              Waypoint Sacar_P2: TCP in base x=-1173.973 y=-367.221 z=3.618 mm, rx=2.0094 ry=-2.4021 rz=-0.0129 rad; joints [10.662, -31.588, 47.899, -16.562, 101.711, 0.111] deg
            Wait Sleep waitTime=0.5
            MoveDirectionNode (selectedDirection=YPlus toolParams=0.0013, 2.0E-4)
              Until TOOL_CONTACT_DETECTION (allowActions=false retraction=0 decelerationAcceleration=9 decelerationAngularAcceleration=34.906585)
            Wait Sleep waitTime=2
            P2 := pose_add(get_actual_tcp_pose(), P2)
            muestrasTomadas := muestrasTomadas+1
          muestrasTomadas := 0
          var_1 := (P2[0])/muestras
          var_2 := (P2[1])/muestras
          rotaciones := get_actual_tcp_pose()
          var_3 := rotaciones[3]
          var_4 := rotaciones[4]
          var_5 := rotaciones[5]
          P2 := p[var_1,var_2,-0.37,var_3,var_4,var_5]
        MoveJ speed 60 deg/s, acceleration 80 deg/s^2 (useActiveTCP=true) feature=Base
          Waypoint Casa2: TCP in base x=-771.144 y=-432.919 z=130.536 mm, rx=2.0101 ry=-2.4029 rz=-0.0102 rad; joints [21.813, -67.428, 96.538, -29.271, 112.826, 0.127] deg
        Folder m1
          var_1 := (P1[0])
          var_2 := (P1[1])
          var_3 := (P2[0])
          var_4 := (P2[1])
          m1 := (var_4-var_2)/(var_3-var_1)
        Folder b1
          b1 := ((m1*var_1)-var_2)*(-1)
        MoveJ speed 60 deg/s, acceleration 80 deg/s^2 (useActiveTCP=true) feature=Base
          Waypoint Casa1: TCP in base x=-416.709 y=-228.23 z=81.827 mm, rx=2.012 ry=-2.4053 rz=-0.0107 rad; joints [11.287, -103.558, 142.129, -38.591, 102.295, 0.04] deg
        Folder P3
          Loop While (checkContinuously=false) expression=muestrasTomadas<muestras
            MoveJ speed 60 deg/s, acceleration 80 deg/s^2 (useActiveTCP=true) feature=Base
              Waypoint Sacar_P3: motionParameters(jointSpeed=1.047198 jointAcceleration=1.396263 cartesianSpeed=0.1 cartesianAcceleration=0.15); TCP in base x=-387.702 y=-99.027 z=-5.945 mm, rx=2.01 ry=-2.4029 rz=-0.0102 rad; joints [-19.937, -108.067, 157.062, -49.107, 71.061, 0.231] deg
            Wait Sleep waitTime=0.5
            MoveDirectionNode (selectedDirection=XPlus toolParams=0.0013, 2.0E-4)
              Until TOOL_CONTACT_DETECTION (allowActions=false retraction=0 decelerationAcceleration=9 decelerationAngularAcceleration=34.906585)
            Wait Sleep waitTime=2
            P3 := pose_add(get_actual_tcp_pose(), P3)
            muestrasTomadas := muestrasTomadas+1
          muestrasTomadas := 0
          var_1 := (P3[0])/muestras
          var_2 := (P3[1])/muestras
          rotaciones := get_actual_tcp_pose()
          var_3 := rotaciones[3]
          var_4 := rotaciones[4]
          var_5 := rotaciones[5]
          P3 := p[var_1,var_2,-0.37,var_3,var_4,var_5]
        MoveJ speed 60 deg/s, acceleration 80 deg/s^2 (useActiveTCP=true) feature=Base
          Waypoint Casa1: TCP in base x=-416.709 y=-228.23 z=81.827 mm, rx=2.012 ry=-2.4053 rz=-0.0107 rad; joints [11.287, -103.558, 142.129, -38.591, 102.295, 0.04] deg
        Folder P4
          Loop While (checkContinuously=false) expression=muestrasTomadas<muestras
            MoveJ speed 60 deg/s, acceleration 80 deg/s^2 (useActiveTCP=true) feature=Base
              Waypoint Sacar_P4: motionParameters(jointSpeed=1.047198 jointAcceleration=1.396263 cartesianSpeed=0.1 cartesianAcceleration=0.15); TCP in base x=-386.694 y=-336.624 z=-4.009 mm, rx=2.0101 ry=-2.4029 rz=-0.0102 rad; joints [30.346, -87.141, 140.524, -53.547, 121.328, 0.136] deg
            Wait Sleep waitTime=0.5
            MoveDirectionNode (selectedDirection=XPlus toolParams=0.0013, 2.0E-4)
              Until TOOL_CONTACT_DETECTION (allowActions=false retraction=0 decelerationAcceleration=9 decelerationAngularAcceleration=34.906585)
            Wait Sleep waitTime=2
            P4 := pose_add(get_actual_tcp_pose(), P4)
            muestrasTomadas := muestrasTomadas+1
          muestrasTomadas := 0
          var_1 := (P4[0])/muestras
          var_2 := (P4[1])/muestras
          rotaciones := get_actual_tcp_pose()
          var_3 := rotaciones[3]
          var_4 := rotaciones[4]
          var_5 := rotaciones[5]
          P4 := p[var_1,var_2,-0.37,var_3,var_4,var_5]
        MoveJ speed 60 deg/s, acceleration 80 deg/s^2 (useActiveTCP=true) feature=Base
          Waypoint Casa1: TCP in base x=-416.709 y=-228.23 z=81.827 mm, rx=2.012 ry=-2.4053 rz=-0.0107 rad; joints [11.287, -103.558, 142.129, -38.591, 102.295, 0.04] deg
        Folder m2
          var_1 := (P3[0])
          var_2 := (P3[1])
          var_3 := (P4[0])
          var_4 := (P4[1])
          m2 := (var_4-var_2)/(var_3-var_1)
        Folder b2
          b2 := ((m2*var_1)-var_2)*(-1)
        Folder Xd y Yd
          Xd := (b2-b1)/(m1-m2)
          Yd := (m1*Xd)+b1
        Folder Xp y Yp
          Xp := (1)/(sqrt((m1*m1)+1))
          Yp := (m2)/(sqrt((m2*m2)+1))
        Folder Origen
          Xfin := ((0*Xp)-(Xd)-(0*(1/m2)))*(-1)
          Yfin := ((0*Yp)-(Yd)+(0*m1))*(-1)
          rotaciones := get_actual_tcp_pose()
          var_3 := rotaciones[3]
          var_4 := rotaciones[4]
          var_5 := rotaciones[5]
          PosFinal := p[Xfin+0.00208915,Yfin+0.00208915,0.11,var_3,var_4,var_5]
          origen := PosFinal
        MoveJ speed 60 deg/s, acceleration 80 deg/s^2 (useActiveTCP=true) feature=Base
          Waypoint Waypoint (Variable): motionParameters(jointSpeed=1.047198 jointAcceleration=1.396263 cartesianSpeed=0.15 cartesianAcceleration=0.2); variable=PosFinal
        MoveDirectionNode (selectedDirection=ZPlus)
          Until DISTANCE (allowActions=false deceleration=3 distanceNodeType=STOP) Distance=0.1; motionParameters(blendRadius=0)
        MoveJ speed 60 deg/s, acceleration 80 deg/s^2 (useActiveTCP=true) feature=Base
          Waypoint Casa2: TCP in base x=-771.144 y=-432.919 z=130.536 mm, rx=2.0101 ry=-2.4029 rz=-0.0102 rad; joints [21.813, -67.428, 96.538, -29.271, 112.826, 0.127] deg
        Folder Linea1
          SuppressedNode
            Folder Buje1
              Xfin := ((0.09525*Xp)-(Xd)-(-0.0127*(1/m2)))*(-1)
              Yfin := ((-0.0127*Yp)-(Yd)+(0.09525*m1))*(-1)
              rotaciones := get_actual_tcp_pose()
              var_3 := rotaciones[3]
              var_4 := rotaciones[4]
              var_5 := rotaciones[5]
              PosFinal := p[Xfin+0.00208915,Yfin+0.00208915,0.03,var_3,var_4,var_5]
              MoveL speed 250 mm/s, acceleration 1200 mm/s^2 (useActiveTCP=true) feature=Base
                MoveJ speed 60 deg/s, acceleration 80 deg/s^2 (useActiveTCP=true) feature=Base
                  Waypoint Waypoint (Variable): motionParameters(jointSpeed=1.047198 jointAcceleration=1.396263 cartesianSpeed=0.15 cartesianAcceleration=0.2); variable=PosFinal
                MoveDirectionNode (selectedDirection=ZMinus toolParams=0.02, 0.02)
                  Until DISTANCE (allowActions=false deceleration=3 distanceNodeType=STOP) Distance=0.035; motionParameters(blendRadius=0)
                MoveDirectionNode (selectedDirection=ZPlus toolParams=0.02, 0.02)
                  Until DISTANCE (allowActions=false deceleration=3 distanceNodeType=STOP) Distance=0.035; motionParameters(blendRadius=0)
          SuppressedNode
            Folder Buje2
              Xfin := ((0.12065*Xp)-(Xd)-(-0.0127*(1/m2)))*(-1)
              Yfin := ((-0.0127*Yp)-(Yd)+(0.12065*m1))*(-1)
              rotaciones := get_actual_tcp_pose()
              var_3 := rotaciones[3]
              var_4 := rotaciones[4]
              var_5 := rotaciones[5]
              PosFinal := p[Xfin+0.00208915,Yfin+0.00208915,0.03,var_3,var_4,var_5]
              MoveL speed 250 mm/s, acceleration 1200 mm/s^2 (useActiveTCP=true) feature=Base
                MoveJ speed 60 deg/s, acceleration 80 deg/s^2 (useActiveTCP=true) feature=Base
                  Waypoint Waypoint (Variable): motionParameters(jointSpeed=1.047198 jointAcceleration=1.396263 cartesianSpeed=0.15 cartesianAcceleration=0.2); variable=PosFinal
                MoveDirectionNode (selectedDirection=ZMinus toolParams=0.02, 0.02)
                  Until DISTANCE (allowActions=false deceleration=3 distanceNodeType=STOP) Distance=0.035; motionParameters(blendRadius=0)
                MoveDirectionNode (selectedDirection=ZPlus toolParams=0.02, 0.02)
                  Until DISTANCE (allowActions=false deceleration=3 distanceNodeType=STOP) Distance=0.035; motionParameters(blendRadius=0)
          SuppressedNode
            Folder Buje3
              Xfin := ((0.14605*Xp)-(Xd)-(-0.0127*(1/m2)))*(-1)
              Yfin := ((-0.0127*Yp)-(Yd)+(0.14605*m1))*(-1)
              rotaciones := get_actual_tcp_pose()
              var_3 := rotaciones[3]
              var_4 := rotaciones[4]
              var_5 := rotaciones[5]
              PosFinal := p[Xfin+0.00208915,Yfin+0.00208915,0.03,var_3,var_4,var_5]
              MoveL speed 250 mm/s, acceleration 1200 mm/s^2 (useActiveTCP=true) feature=Base
                MoveJ speed 60 deg/s, acceleration 80 deg/s^2 (useActiveTCP=true) feature=Base
                  Waypoint Waypoint (Variable): motionParameters(jointSpeed=1.047198 jointAcceleration=1.396263 cartesianSpeed=0.15 cartesianAcceleration=0.2); variable=PosFinal
                MoveDirectionNode (selectedDirection=ZMinus toolParams=0.02, 0.02)
                  Until DISTANCE (allowActions=false deceleration=3 distanceNodeType=STOP) Distance=0.035; motionParameters(blendRadius=0)
                MoveDirectionNode (selectedDirection=ZPlus toolParams=0.02, 0.02)
                  Until DISTANCE (allowActions=false deceleration=3 distanceNodeType=STOP) Distance=0.035; motionParameters(blendRadius=0)
          SuppressedNode
            Folder Buje4
              Xfin := ((0.17145*Xp)-(Xd)-(-0.0127*(1/m2)))*(-1)
              Yfin := ((-0.0127*Yp)-(Yd)+(0.17145*m1))*(-1)
              rotaciones := get_actual_tcp_pose()
              var_3 := rotaciones[3]
              var_4 := rotaciones[4]
              var_5 := rotaciones[5]
              PosFinal := p[Xfin+0.00208915,Yfin+0.00208915,0.03,var_3,var_4,var_5]
              MoveL speed 250 mm/s, acceleration 1200 mm/s^2 (useActiveTCP=true) feature=Base
                MoveJ speed 60 deg/s, acceleration 80 deg/s^2 (useActiveTCP=true) feature=Base
                  Waypoint Waypoint (Variable): motionParameters(jointSpeed=1.047198 jointAcceleration=1.396263 cartesianSpeed=0.15 cartesianAcceleration=0.2); variable=PosFinal
                MoveDirectionNode (selectedDirection=ZMinus toolParams=0.02, 0.02)
                  Until DISTANCE (allowActions=false deceleration=3 distanceNodeType=STOP) Distance=0.035; motionParameters(blendRadius=0)
                MoveDirectionNode (selectedDirection=ZPlus toolParams=0.02, 0.02)
                  Until DISTANCE (allowActions=false deceleration=3 distanceNodeType=STOP) Distance=0.035; motionParameters(blendRadius=0)
          SuppressedNode
            Folder Buje5
              Xfin := ((0.19685*Xp)-(Xd)-(-0.0127*(1/m2)))*(-1)
              Yfin := ((-0.0127*Yp)-(Yd)+(0.19685*m1))*(-1)
              rotaciones := get_actual_tcp_pose()
              var_3 := rotaciones[3]
              var_4 := rotaciones[4]
              var_5 := rotaciones[5]
              PosFinal := p[Xfin+0.00208915,Yfin+0.00208915,0.03,var_3,var_4,var_5]
              MoveL speed 250 mm/s, acceleration 1200 mm/s^2 (useActiveTCP=true) feature=Base
                MoveJ speed 60 deg/s, acceleration 80 deg/s^2 (useActiveTCP=true) feature=Base
                  Waypoint Waypoint (Variable): motionParameters(jointSpeed=1.047198 jointAcceleration=1.396263 cartesianSpeed=0.15 cartesianAcceleration=0.2); variable=PosFinal
                MoveDirectionNode (selectedDirection=ZMinus toolParams=0.02, 0.02)
                  Until DISTANCE (allowActions=false deceleration=3 distanceNodeType=STOP) Distance=0.035; motionParameters(blendRadius=0)
                MoveDirectionNode (selectedDirection=ZPlus toolParams=0.02, 0.02)
                  Until DISTANCE (allowActions=false deceleration=3 distanceNodeType=STOP) Distance=0.035; motionParameters(blendRadius=0)
          SuppressedNode
            Folder Buje6
              Xfin := ((0.22225*Xp)-(Xd)-(-0.0127*(1/m2)))*(-1)
              Yfin := ((-0.0127*Yp)-(Yd)+(0.22225*m1))*(-1)
              rotaciones := get_actual_tcp_pose()
              var_3 := rotaciones[3]
              var_4 := rotaciones[4]
              var_5 := rotaciones[5]
              PosFinal := p[Xfin+0.00208915,Yfin+0.00208915,0.03,var_3,var_4,var_5]
              MoveL speed 250 mm/s, acceleration 1200 mm/s^2 (useActiveTCP=true) feature=Base
                MoveJ speed 60 deg/s, acceleration 80 deg/s^2 (useActiveTCP=true) feature=Base
                  Waypoint Waypoint (Variable): motionParameters(jointSpeed=1.047198 jointAcceleration=1.396263 cartesianSpeed=0.15 cartesianAcceleration=0.2); variable=PosFinal
                MoveDirectionNode (selectedDirection=ZMinus toolParams=0.02, 0.02)
                  Until DISTANCE (allowActions=false deceleration=3 distanceNodeType=STOP) Distance=0.035; motionParameters(blendRadius=0)
                MoveDirectionNode (selectedDirection=ZPlus toolParams=0.02, 0.02)
                  Until DISTANCE (allowActions=false deceleration=3 distanceNodeType=STOP) Distance=0.035; motionParameters(blendRadius=0)
          SuppressedNode
            Folder Buje7
              Xfin := ((0.24765*Xp)-(Xd)-(-0.0127*(1/m2)))*(-1)
              Yfin := ((-0.0127*Yp)-(Yd)+(0.24765*m1))*(-1)
              rotaciones := get_actual_tcp_pose()
              var_3 := rotaciones[3]
              var_4 := rotaciones[4]
              var_5 := rotaciones[5]
              PosFinal := p[Xfin+0.00208915,Yfin+0.00208915,0.03,var_3,var_4,var_5]
              MoveL speed 250 mm/s, acceleration 1200 mm/s^2 (useActiveTCP=true) feature=Base
                MoveJ speed 60 deg/s, acceleration 80 deg/s^2 (useActiveTCP=true) feature=Base
                  Waypoint Waypoint (Variable): motionParameters(jointSpeed=1.047198 jointAcceleration=1.396263 cartesianSpeed=0.15 cartesianAcceleration=0.2); variable=PosFinal
                MoveDirectionNode (selectedDirection=ZMinus toolParams=0.02, 0.02)
                  Until DISTANCE (allowActions=false deceleration=3 distanceNodeType=STOP) Distance=0.035; motionParameters(blendRadius=0)
                MoveDirectionNode (selectedDirection=ZPlus toolParams=0.02, 0.02)
                  Until DISTANCE (allowActions=false deceleration=3 distanceNodeType=STOP) Distance=0.035; motionParameters(blendRadius=0)
          SuppressedNode
            Folder Buje8
              Xfin := ((0.27305*Xp)-(Xd)-(-0.0127*(1/m2)))*(-1)
              Yfin := ((-0.0127*Yp)-(Yd)+(0.27305*m1))*(-1)
              rotaciones := get_actual_tcp_pose()
              var_3 := rotaciones[3]
              var_4 := rotaciones[4]
              var_5 := rotaciones[5]
              PosFinal := p[Xfin+0.00208915,Yfin+0.00208915,0.03,var_3,var_4,var_5]
              MoveL speed 250 mm/s, acceleration 1200 mm/s^2 (useActiveTCP=true) feature=Base
                MoveJ speed 60 deg/s, acceleration 80 deg/s^2 (useActiveTCP=true) feature=Base
                  Waypoint Waypoint (Variable): motionParameters(jointSpeed=1.047198 jointAcceleration=1.396263 cartesianSpeed=0.15 cartesianAcceleration=0.2); variable=PosFinal
                MoveDirectionNode (selectedDirection=ZMinus toolParams=0.02, 0.02)
                  Until DISTANCE (allowActions=false deceleration=3 distanceNodeType=STOP) Distance=0.035; motionParameters(blendRadius=0)
                MoveDirectionNode (selectedDirection=ZPlus toolParams=0.02, 0.02)
                  Until DISTANCE (allowActions=false deceleration=3 distanceNodeType=STOP) Distance=0.035; motionParameters(blendRadius=0)
          SuppressedNode
            Folder Buje9
              Xfin := ((0.29845*Xp)-(Xd)-(-0.0127*(1/m2)))*(-1)
              Yfin := ((-0.0127*Yp)-(Yd)+(0.29845*m1))*(-1)
              rotaciones := get_actual_tcp_pose()
              var_3 := rotaciones[3]
              var_4 := rotaciones[4]
              var_5 := rotaciones[5]
              PosFinal := p[Xfin+0.00208915,Yfin+0.00208915,0.03,var_3,var_4,var_5]
              MoveL speed 250 mm/s, acceleration 1200 mm/s^2 (useActiveTCP=true) feature=Base
                MoveJ speed 60 deg/s, acceleration 80 deg/s^2 (useActiveTCP=true) feature=Base
                  Waypoint Waypoint (Variable): motionParameters(jointSpeed=1.047198 jointAcceleration=1.396263 cartesianSpeed=0.15 cartesianAcceleration=0.2); variable=PosFinal
                MoveDirectionNode (selectedDirection=ZMinus toolParams=0.02, 0.02)
                  Until DISTANCE (allowActions=false deceleration=3 distanceNodeType=STOP) Distance=0.035; motionParameters(blendRadius=0)
                MoveDirectionNode (selectedDirection=ZPlus toolParams=0.02, 0.02)
                  Until DISTANCE (allowActions=false deceleration=3 distanceNodeType=STOP) Distance=0.035; motionParameters(blendRadius=0)
          SuppressedNode
            Folder Buje10
              Xfin := ((0.32385*Xp)-(Xd)-(-0.0127*(1/m2)))*(-1)
              Yfin := ((-0.0127*Yp)-(Yd)+(0.32385*m1))*(-1)
              rotaciones := get_actual_tcp_pose()
              var_3 := rotaciones[3]
              var_4 := rotaciones[4]
              var_5 := rotaciones[5]
              PosFinal := p[Xfin+0.00208915,Yfin+0.00208915,0.03,var_3,var_4,var_5]
              MoveL speed 250 mm/s, acceleration 1200 mm/s^2 (useActiveTCP=true) feature=Base
                MoveJ speed 60 deg/s, acceleration 80 deg/s^2 (useActiveTCP=true) feature=Base
                  Waypoint Waypoint (Variable): motionParameters(jointSpeed=1.047198 jointAcceleration=1.396263 cartesianSpeed=0.15 cartesianAcceleration=0.2); variable=PosFinal
                MoveDirectionNode (selectedDirection=ZMinus toolParams=0.02, 0.02)
                  Until DISTANCE (allowActions=false deceleration=3 distanceNodeType=STOP) Distance=0.035; motionParameters(blendRadius=0)
                MoveDirectionNode (selectedDirection=ZPlus toolParams=0.02, 0.02)
                  Until DISTANCE (allowActions=false deceleration=3 distanceNodeType=STOP) Distance=0.035; motionParameters(blendRadius=0)
          SuppressedNode
            Folder Buje11
              Xfin := ((0.34925*Xp)-(Xd)-(-0.0127*(1/m2)))*(-1)
              Yfin := ((-0.0127*Yp)-(Yd)+(0.34925*m1))*(-1)
              rotaciones := get_actual_tcp_pose()
              var_3 := rotaciones[3]
              var_4 := rotaciones[4]
              var_5 := rotaciones[5]
              PosFinal := p[Xfin+0.00208915,Yfin+0.00208915,0.03,var_3,var_4,var_5]
              MoveL speed 250 mm/s, acceleration 1200 mm/s^2 (useActiveTCP=true) feature=Base
                MoveJ speed 60 deg/s, acceleration 80 deg/s^2 (useActiveTCP=true) feature=Base
                  Waypoint Waypoint (Variable): motionParameters(jointSpeed=1.047198 jointAcceleration=1.396263 cartesianSpeed=0.15 cartesianAcceleration=0.2); variable=PosFinal
                MoveDirectionNode (selectedDirection=ZMinus toolParams=0.02, 0.02)
                  Until DISTANCE (allowActions=false deceleration=3 distanceNodeType=STOP) Distance=0.035; motionParameters(blendRadius=0)
                MoveDirectionNode (selectedDirection=ZPlus toolParams=0.02, 0.02)
                  Until DISTANCE (allowActions=false deceleration=3 distanceNodeType=STOP) Distance=0.035; motionParameters(blendRadius=0)
          SuppressedNode
            Folder Buje12
              Xfin := ((0.37465*Xp)-(Xd)-(-0.0127*(1/m2)))*(-1)
              Yfin := ((-0.0127*Yp)-(Yd)+(0.37465*m1))*(-1)
              rotaciones := get_actual_tcp_pose()
              var_3 := rotaciones[3]
              var_4 := rotaciones[4]
              var_5 := rotaciones[5]
              PosFinal := p[Xfin+0.00208915,Yfin+0.00208915,0.03,var_3,var_4,var_5]
              MoveL speed 250 mm/s, acceleration 1200 mm/s^2 (useActiveTCP=true) feature=Base
                MoveJ speed 60 deg/s, acceleration 80 deg/s^2 (useActiveTCP=true) feature=Base
                  Waypoint Waypoint (Variable): motionParameters(jointSpeed=1.047198 jointAcceleration=1.396263 cartesianSpeed=0.15 cartesianAcceleration=0.2); variable=PosFinal
                MoveDirectionNode (selectedDirection=ZMinus toolParams=0.02, 0.02)
                  Until DISTANCE (allowActions=false deceleration=3 distanceNodeType=STOP) Distance=0.035; motionParameters(blendRadius=0)
                MoveDirectionNode (selectedDirection=ZPlus toolParams=0.02, 0.02)
                  Until DISTANCE (allowActions=false deceleration=3 distanceNodeType=STOP) Distance=0.035; motionParameters(blendRadius=0)
          SuppressedNode
            Folder Buje13
              Xfin := ((0.40005*Xp)-(Xd)-(-0.0127*(1/m2)))*(-1)
              Yfin := ((-0.0127*Yp)-(Yd)+(0.40005*m1))*(-1)
              rotaciones := get_actual_tcp_pose()
              var_3 := rotaciones[3]
              var_4 := rotaciones[4]
              var_5 := rotaciones[5]
              PosFinal := p[Xfin+0.00208915,Yfin+0.00208915,0.03,var_3,var_4,var_5]
              MoveL speed 250 mm/s, acceleration 1200 mm/s^2 (useActiveTCP=true) feature=Base
                MoveJ speed 60 deg/s, acceleration 80 deg/s^2 (useActiveTCP=true) feature=Base
                  Waypoint Waypoint (Variable): motionParameters(jointSpeed=1.047198 jointAcceleration=1.396263 cartesianSpeed=0.15 cartesianAcceleration=0.2); variable=PosFinal
                MoveDirectionNode (selectedDirection=ZMinus toolParams=0.02, 0.02)
                  Until DISTANCE (allowActions=false deceleration=3 distanceNodeType=STOP) Distance=0.035; motionParameters(blendRadius=0)
                MoveDirectionNode (selectedDirection=ZPlus toolParams=0.02, 0.02)
                  Until DISTANCE (allowActions=false deceleration=3 distanceNodeType=STOP) Distance=0.035; motionParameters(blendRadius=0)
          SuppressedNode
            Folder Buje14
              Xfin := ((0.42545*Xp)-(Xd)-(-0.0127*(1/m2)))*(-1)
              Yfin := ((-0.0127*Yp)-(Yd)+(0.42545*m1))*(-1)
              rotaciones := get_actual_tcp_pose()
              var_3 := rotaciones[3]
              var_4 := rotaciones[4]
              var_5 := rotaciones[5]
              PosFinal := p[Xfin+0.00208915,Yfin+0.00208915,0.03,var_3,var_4,var_5]
              MoveL speed 250 mm/s, acceleration 1200 mm/s^2 (useActiveTCP=true) feature=Base
                MoveJ speed 60 deg/s, acceleration 80 deg/s^2 (useActiveTCP=true) feature=Base
                  Waypoint Waypoint (Variable): motionParameters(jointSpeed=1.047198 jointAcceleration=1.396263 cartesianSpeed=0.15 cartesianAcceleration=0.2); variable=PosFinal
                MoveDirectionNode (selectedDirection=ZMinus toolParams=0.02, 0.02)
                  Until DISTANCE (allowActions=false deceleration=3 distanceNodeType=STOP) Distance=0.035; motionParameters(blendRadius=0)
                MoveDirectionNode (selectedDirection=ZPlus toolParams=0.02, 0.02)
                  Until DISTANCE (allowActions=false deceleration=3 distanceNodeType=STOP) Distance=0.035; motionParameters(blendRadius=0)
          SuppressedNode
            Folder Buje15
              Xfin := ((0.45085*Xp)-(Xd)-(-0.0127*(1/m2)))*(-1)
              Yfin := ((-0.0127*Yp)-(Yd)+(0.45085*m1))*(-1)
              rotaciones := get_actual_tcp_pose()
              var_3 := rotaciones[3]
              var_4 := rotaciones[4]
              var_5 := rotaciones[5]
              PosFinal := p[Xfin+0.00208915,Yfin+0.00208915,0.03,var_3,var_4,var_5]
              MoveL speed 250 mm/s, acceleration 1200 mm/s^2 (useActiveTCP=true) feature=Base
                MoveJ speed 60 deg/s, acceleration 80 deg/s^2 (useActiveTCP=true) feature=Base
                  Waypoint Waypoint (Variable): motionParameters(jointSpeed=1.047198 jointAcceleration=1.396263 cartesianSpeed=0.15 cartesianAcceleration=0.2); variable=PosFinal
                MoveDirectionNode (selectedDirection=ZMinus toolParams=0.02, 0.02)
                  Until DISTANCE (allowActions=false deceleration=3 distanceNodeType=STOP) Distance=0.035; motionParameters(blendRadius=0)
                MoveDirectionNode (selectedDirection=ZPlus toolParams=0.02, 0.02)
                  Until DISTANCE (allowActions=false deceleration=3 distanceNodeType=STOP) Distance=0.035; motionParameters(blendRadius=0)
          SuppressedNode
            Folder Buje16
              Xfin := ((0.47625*Xp)-(Xd)-(-0.0127*(1/m2)))*(-1)
              Yfin := ((-0.0127*Yp)-(Yd)+(0.47625*m1))*(-1)
              rotaciones := get_actual_tcp_pose()
              var_3 := rotaciones[3]
              var_4 := rotaciones[4]
              var_5 := rotaciones[5]
              PosFinal := p[Xfin+0.00208915,Yfin+0.00208915,0.03,var_3,var_4,var_5]
              MoveL speed 250 mm/s, acceleration 1200 mm/s^2 (useActiveTCP=true) feature=Base
                MoveJ speed 60 deg/s, acceleration 80 deg/s^2 (useActiveTCP=true) feature=Base
                  Waypoint Waypoint (Variable): motionParameters(jointSpeed=1.047198 jointAcceleration=1.396263 cartesianSpeed=0.15 cartesianAcceleration=0.2); variable=PosFinal
                MoveDirectionNode (selectedDirection=ZMinus toolParams=0.02, 0.02)
                  Until DISTANCE (allowActions=false deceleration=3 distanceNodeType=STOP) Distance=0.035; motionParameters(blendRadius=0)
                MoveDirectionNode (selectedDirection=ZPlus toolParams=0.02, 0.02)
                  Until DISTANCE (allowActions=false deceleration=3 distanceNodeType=STOP) Distance=0.035; motionParameters(blendRadius=0)
          SuppressedNode
            Folder Buje17
              Xfin := ((0.50165*Xp)-(Xd)-(-0.0127*(1/m2)))*(-1)
              Yfin := ((-0.0127*Yp)-(Yd)+(0.50165*m1))*(-1)
              rotaciones := get_actual_tcp_pose()
              var_3 := rotaciones[3]
              var_4 := rotaciones[4]
              var_5 := rotaciones[5]
              PosFinal := p[Xfin+0.00208915,Yfin+0.00208915,0.03,var_3,var_4,var_5]
              MoveL speed 250 mm/s, acceleration 1200 mm/s^2 (useActiveTCP=true) feature=Base
                MoveJ speed 60 deg/s, acceleration 80 deg/s^2 (useActiveTCP=true) feature=Base
                  Waypoint Waypoint (Variable): motionParameters(jointSpeed=1.047198 jointAcceleration=1.396263 cartesianSpeed=0.15 cartesianAcceleration=0.2); variable=PosFinal
                MoveDirectionNode (selectedDirection=ZMinus toolParams=0.02, 0.02)
                  Until DISTANCE (allowActions=false deceleration=3 distanceNodeType=STOP) Distance=0.035; motionParameters(blendRadius=0)
                MoveDirectionNode (selectedDirection=ZPlus toolParams=0.02, 0.02)
                  Until DISTANCE (allowActions=false deceleration=3 distanceNodeType=STOP) Distance=0.035; motionParameters(blendRadius=0)
          SuppressedNode
            Folder Buje18
              Xfin := ((0.52705*Xp)-(Xd)-(-0.0127*(1/m2)))*(-1)
              Yfin := ((-0.0127*Yp)-(Yd)+(0.52705*m1))*(-1)
              rotaciones := get_actual_tcp_pose()
              var_3 := rotaciones[3]
              var_4 := rotaciones[4]
              var_5 := rotaciones[5]
              PosFinal := p[Xfin+0.00208915,Yfin+0.00208915,0.03,var_3,var_4,var_5]
              MoveL speed 250 mm/s, acceleration 1200 mm/s^2 (useActiveTCP=true) feature=Base
                MoveJ speed 60 deg/s, acceleration 80 deg/s^2 (useActiveTCP=true) feature=Base
                  Waypoint Waypoint (Variable): motionParameters(jointSpeed=1.047198 jointAcceleration=1.396263 cartesianSpeed=0.15 cartesianAcceleration=0.2); variable=PosFinal
                MoveDirectionNode (selectedDirection=ZMinus toolParams=0.02, 0.02)
                  Until DISTANCE (allowActions=false deceleration=3 distanceNodeType=STOP) Distance=0.035; motionParameters(blendRadius=0)
                MoveDirectionNode (selectedDirection=ZPlus toolParams=0.02, 0.02)
                  Until DISTANCE (allowActions=false deceleration=3 distanceNodeType=STOP) Distance=0.035; motionParameters(blendRadius=0)
          SuppressedNode
            Folder Buje19
              Xfin := ((0.55245*Xp)-(Xd)-(-0.0127*(1/m2)))*(-1)
              Yfin := ((-0.0127*Yp)-(Yd)+(0.55245*m1))*(-1)
              rotaciones := get_actual_tcp_pose()
              var_3 := rotaciones[3]
              var_4 := rotaciones[4]
              var_5 := rotaciones[5]
              PosFinal := p[Xfin+0.00208915,Yfin+0.00208915,0.03,var_3,var_4,var_5]
              MoveL speed 250 mm/s, acceleration 1200 mm/s^2 (useActiveTCP=true) feature=Base
                MoveJ speed 60 deg/s, acceleration 80 deg/s^2 (useActiveTCP=true) feature=Base
                  Waypoint Waypoint (Variable): motionParameters(jointSpeed=1.047198 jointAcceleration=1.396263 cartesianSpeed=0.15 cartesianAcceleration=0.2); variable=PosFinal
                MoveDirectionNode (selectedDirection=ZMinus toolParams=0.02, 0.02)
                  Until DISTANCE (allowActions=false deceleration=3 distanceNodeType=STOP) Distance=0.035; motionParameters(blendRadius=0)
                MoveDirectionNode (selectedDirection=ZPlus toolParams=0.02, 0.02)
                  Until DISTANCE (allowActions=false deceleration=3 distanceNodeType=STOP) Distance=0.035; motionParameters(blendRadius=0)
          SuppressedNode
            Folder Buje20
              Xfin := ((0.57785*Xp)-(Xd)-(-0.0127*(1/m2)))*(-1)
              Yfin := ((-0.0127*Yp)-(Yd)+(0.57785*m1))*(-1)
              rotaciones := get_actual_tcp_pose()
              var_3 := rotaciones[3]
              var_4 := rotaciones[4]
              var_5 := rotaciones[5]
              PosFinal := p[Xfin+0.00208915,Yfin+0.00208915,0.03,var_3,var_4,var_5]
              MoveL speed 250 mm/s, acceleration 1200 mm/s^2 (useActiveTCP=true) feature=Base
                MoveJ speed 60 deg/s, acceleration 80 deg/s^2 (useActiveTCP=true) feature=Base
                  Waypoint Waypoint (Variable): motionParameters(jointSpeed=1.047198 jointAcceleration=1.396263 cartesianSpeed=0.15 cartesianAcceleration=0.2); variable=PosFinal
                MoveDirectionNode (selectedDirection=ZMinus toolParams=0.02, 0.02)
                  Until DISTANCE (allowActions=false deceleration=3 distanceNodeType=STOP) Distance=0.035; motionParameters(blendRadius=0)
                MoveDirectionNode (selectedDirection=ZPlus toolParams=0.02, 0.02)
                  Until DISTANCE (allowActions=false deceleration=3 distanceNodeType=STOP) Distance=0.035; motionParameters(blendRadius=0)
          SuppressedNode
            Folder Buje21
              Xfin := ((0.60325*Xp)-(Xd)-(-0.0127*(1/m2)))*(-1)
              Yfin := ((-0.0127*Yp)-(Yd)+(0.60325*m1))*(-1)
              rotaciones := get_actual_tcp_pose()
              var_3 := rotaciones[3]
              var_4 := rotaciones[4]
              var_5 := rotaciones[5]
              PosFinal := p[Xfin+0.00208915,Yfin+0.00208915,0.03,var_3,var_4,var_5]
              MoveL speed 250 mm/s, acceleration 1200 mm/s^2 (useActiveTCP=true) feature=Base
                MoveJ speed 60 deg/s, acceleration 80 deg/s^2 (useActiveTCP=true) feature=Base
                  Waypoint Waypoint (Variable): motionParameters(jointSpeed=1.047198 jointAcceleration=1.396263 cartesianSpeed=0.15 cartesianAcceleration=0.2); variable=PosFinal
                MoveDirectionNode (selectedDirection=ZMinus toolParams=0.02, 0.02)
                  Until DISTANCE (allowActions=false deceleration=3 distanceNodeType=STOP) Distance=0.035; motionParameters(blendRadius=0)
                MoveDirectionNode (selectedDirection=ZPlus toolParams=0.02, 0.02)
                  Until DISTANCE (allowActions=false deceleration=3 distanceNodeType=STOP) Distance=0.035; motionParameters(blendRadius=0)
          SuppressedNode
            Folder Buje22
              Xfin := ((0.62865*Xp)-(Xd)-(-0.0127*(1/m2)))*(-1)
              Yfin := ((-0.0127*Yp)-(Yd)+(0.62865*m1))*(-1)
              rotaciones := get_actual_tcp_pose()
              var_3 := rotaciones[3]
              var_4 := rotaciones[4]
              var_5 := rotaciones[5]
              PosFinal := p[Xfin+0.00208915,Yfin+0.00208915,0.03,var_3,var_4,var_5]
              MoveL speed 250 mm/s, acceleration 1200 mm/s^2 (useActiveTCP=true) feature=Base
                MoveJ speed 60 deg/s, acceleration 80 deg/s^2 (useActiveTCP=true) feature=Base
                  Waypoint Waypoint (Variable): motionParameters(jointSpeed=1.047198 jointAcceleration=1.396263 cartesianSpeed=0.15 cartesianAcceleration=0.2); variable=PosFinal
                MoveDirectionNode (selectedDirection=ZMinus toolParams=0.02, 0.02)
                  Until DISTANCE (allowActions=false deceleration=3 distanceNodeType=STOP) Distance=0.035; motionParameters(blendRadius=0)
                MoveDirectionNode (selectedDirection=ZPlus toolParams=0.02, 0.02)
                  Until DISTANCE (allowActions=false deceleration=3 distanceNodeType=STOP) Distance=0.035; motionParameters(blendRadius=0)
          SuppressedNode
            Folder Buje23
              Xfin := ((0.65405*Xp)-(Xd)-(-0.0127*(1/m2)))*(-1)
              Yfin := ((-0.0127*Yp)-(Yd)+(0.65405*m1))*(-1)
              rotaciones := get_actual_tcp_pose()
              var_3 := rotaciones[3]
              var_4 := rotaciones[4]
              var_5 := rotaciones[5]
              PosFinal := p[Xfin+0.00208915,Yfin+0.00208915,0.03,var_3,var_4,var_5]
              MoveL speed 250 mm/s, acceleration 1200 mm/s^2 (useActiveTCP=true) feature=Base
                MoveJ speed 60 deg/s, acceleration 80 deg/s^2 (useActiveTCP=true) feature=Base
                  Waypoint Waypoint (Variable): motionParameters(jointSpeed=1.047198 jointAcceleration=1.396263 cartesianSpeed=0.15 cartesianAcceleration=0.2); variable=PosFinal
                MoveDirectionNode (selectedDirection=ZMinus toolParams=0.02, 0.02)
                  Until DISTANCE (allowActions=false deceleration=3 distanceNodeType=STOP) Distance=0.035; motionParameters(blendRadius=0)
                MoveDirectionNode (selectedDirection=ZPlus toolParams=0.02, 0.02)
                  Until DISTANCE (allowActions=false deceleration=3 distanceNodeType=STOP) Distance=0.035; motionParameters(blendRadius=0)
          SuppressedNode
            Folder Buje24
              Xfin := ((0.67945*Xp)-(Xd)-(-0.0127*(1/m2)))*(-1)
              Yfin := ((-0.0127*Yp)-(Yd)+(0.67945*m1))*(-1)
              rotaciones := get_actual_tcp_pose()
              var_3 := rotaciones[3]
              var_4 := rotaciones[4]
              var_5 := rotaciones[5]
              PosFinal := p[Xfin+0.00208915,Yfin+0.00208915,0.03,var_3,var_4,var_5]
              MoveL speed 250 mm/s, acceleration 1200 mm/s^2 (useActiveTCP=true) feature=Base
                MoveJ speed 60 deg/s, acceleration 80 deg/s^2 (useActiveTCP=true) feature=Base
                  Waypoint Waypoint (Variable): motionParameters(jointSpeed=1.047198 jointAcceleration=1.396263 cartesianSpeed=0.15 cartesianAcceleration=0.2); variable=PosFinal
                MoveDirectionNode (selectedDirection=ZMinus toolParams=0.02, 0.02)
                  Until DISTANCE (allowActions=false deceleration=3 distanceNodeType=STOP) Distance=0.035; motionParameters(blendRadius=0)
                MoveDirectionNode (selectedDirection=ZPlus toolParams=0.02, 0.02)
                  Until DISTANCE (allowActions=false deceleration=3 distanceNodeType=STOP) Distance=0.035; motionParameters(blendRadius=0)
          SuppressedNode
            Folder Buje25
              Xfin := ((0.70485*Xp)-(Xd)-(-0.0127*(1/m2)))*(-1)
              Yfin := ((-0.0127*Yp)-(Yd)+(0.70485*m1))*(-1)
              rotaciones := get_actual_tcp_pose()
              var_3 := rotaciones[3]
              var_4 := rotaciones[4]
              var_5 := rotaciones[5]
              PosFinal := p[Xfin+0.00208915,Yfin+0.00208915,0.03,var_3,var_4,var_5]
              MoveL speed 250 mm/s, acceleration 1200 mm/s^2 (useActiveTCP=true) feature=Base
                MoveJ speed 60 deg/s, acceleration 80 deg/s^2 (useActiveTCP=true) feature=Base
                  Waypoint Waypoint (Variable): motionParameters(jointSpeed=1.047198 jointAcceleration=1.396263 cartesianSpeed=0.15 cartesianAcceleration=0.2); variable=PosFinal
                MoveDirectionNode (selectedDirection=ZMinus toolParams=0.02, 0.02)
                  Until DISTANCE (allowActions=false deceleration=3 distanceNodeType=STOP) Distance=0.035; motionParameters(blendRadius=0)
                MoveDirectionNode (selectedDirection=ZPlus toolParams=0.02, 0.02)
                  Until DISTANCE (allowActions=false deceleration=3 distanceNodeType=STOP) Distance=0.035; motionParameters(blendRadius=0)
          SuppressedNode
            Folder Buje26
              Xfin := ((0.73025*Xp)-(Xd)-(-0.0127*(1/m2)))*(-1)
              Yfin := ((-0.0127*Yp)-(Yd)+(0.73025*m1))*(-1)
              rotaciones := get_actual_tcp_pose()
              var_3 := rotaciones[3]
              var_4 := rotaciones[4]
              var_5 := rotaciones[5]
              PosFinal := p[Xfin+0.00208915,Yfin+0.00208915,0.03,var_3,var_4,var_5]
              MoveL speed 250 mm/s, acceleration 1200 mm/s^2 (useActiveTCP=true) feature=Base
                MoveJ speed 60 deg/s, acceleration 80 deg/s^2 (useActiveTCP=true) feature=Base
                  Waypoint Waypoint (Variable): motionParameters(jointSpeed=1.047198 jointAcceleration=1.396263 cartesianSpeed=0.15 cartesianAcceleration=0.2); variable=PosFinal
                MoveDirectionNode (selectedDirection=ZMinus toolParams=0.02, 0.02)
                  Until DISTANCE (allowActions=false deceleration=3 distanceNodeType=STOP) Distance=0.035; motionParameters(blendRadius=0)
                MoveDirectionNode (selectedDirection=ZPlus toolParams=0.02, 0.02)
                  Until DISTANCE (allowActions=false deceleration=3 distanceNodeType=STOP) Distance=0.035; motionParameters(blendRadius=0)
          Folder Buje27
            Xfin := ((0.75565*Xp)-(Xd)-(-0.0127*(1/m2)))*(-1)
            Yfin := ((-0.0127*Yp)-(Yd)+(0.75565*m1))*(-1)
            rotaciones := get_actual_tcp_pose()
            var_3 := rotaciones[3]
            var_4 := rotaciones[4]
            var_5 := rotaciones[5]
            PosFinal := p[Xfin+0.00208915,Yfin+0.00208915,0.03,var_3,var_4,var_5]
            MoveL speed 250 mm/s, acceleration 1200 mm/s^2 (useActiveTCP=true) feature=Base
              MoveJ speed 60 deg/s, acceleration 80 deg/s^2 (useActiveTCP=true) feature=Base
                Waypoint Waypoint (Variable): motionParameters(jointSpeed=1.047198 jointAcceleration=1.396263 cartesianSpeed=0.15 cartesianAcceleration=0.2); variable=PosFinal
              MoveDirectionNode (selectedDirection=ZMinus toolParams=0.02, 0.02)
                Until DISTANCE (allowActions=false deceleration=3 distanceNodeType=STOP) Distance=0.035; motionParameters(blendRadius=0)
              MoveDirectionNode (selectedDirection=ZPlus toolParams=0.02, 0.02)
                Until DISTANCE (allowActions=false deceleration=3 distanceNodeType=STOP) Distance=0.035; motionParameters(blendRadius=0)
          Popup Message (haltProgram=false message=oi inputType=Text)
        MoveJ speed 60 deg/s, acceleration 80 deg/s^2 (useActiveTCP=true) feature=Base
          Waypoint Casa1: TCP in base x=-416.709 y=-228.23 z=81.827 mm, rx=2.012 ry=-2.4053 rz=-0.0107 rad; joints [11.287, -103.558, 142.129, -38.591, 102.295, 0.04] deg
        Folder Buje1
          Xfin := ((0.09525*Xp)-(Xd)-(0.3937*(1/m2)))*(-1)
          Yfin := ((0.3937*Yp)-(Yd)+(0.09525*m1))*(-1)
          rotaciones := get_actual_tcp_pose()
          var_3 := rotaciones[3]
          var_4 := rotaciones[4]
          var_5 := rotaciones[5]
          PosFinal := p[Xfin+0.00208915,Yfin+0.00208915,-0.44,var_3,var_4,var_5]
          MoveL speed 250 mm/s, acceleration 1200 mm/s^2 (useActiveTCP=true) feature=Base
            MoveJ speed 60 deg/s, acceleration 80 deg/s^2 (useActiveTCP=true) feature=Base
              Waypoint Waypoint (Variable): motionParameters(jointSpeed=1.047198 jointAcceleration=1.396263 cartesianSpeed=0.15 cartesianAcceleration=0.2); variable=PosFinal
            MoveDirectionNode (selectedDirection=ZMinus toolParams=0.02, 0.02)
              Until DISTANCE (allowActions=false deceleration=3 distanceNodeType=STOP) Distance=0.075; motionParameters(blendRadius=0)
            MoveDirectionNode (selectedDirection=ZPlus toolParams=0.02, 0.02)
              Until DISTANCE (allowActions=false deceleration=3 distanceNodeType=STOP) Distance=0.075; motionParameters(blendRadius=0)
        Folder Buje2
          Xfin := ((0.12065*Xp)-(Xd)-(0.3937*(1/m2)))*(-1)
          Yfin := ((0.3937*Yp)-(Yd)+(0.12065*m1))*(-1)
          rotaciones := get_actual_tcp_pose()
          var_3 := rotaciones[3]
          var_4 := rotaciones[4]
          var_5 := rotaciones[5]
          PosFinal := p[Xfin+0.00208915,Yfin+0.00208915,-0.44,var_3,var_4,var_5]
          MoveL speed 250 mm/s, acceleration 1200 mm/s^2 (useActiveTCP=true) feature=Base
            MoveJ speed 60 deg/s, acceleration 80 deg/s^2 (useActiveTCP=true) feature=Base
              Waypoint Waypoint (Variable): motionParameters(jointSpeed=1.047198 jointAcceleration=1.396263 cartesianSpeed=0.15 cartesianAcceleration=0.2); variable=PosFinal
            MoveDirectionNode (selectedDirection=ZMinus toolParams=0.02, 0.02)
              Until DISTANCE (allowActions=false deceleration=3 distanceNodeType=STOP) Distance=0.075; motionParameters(blendRadius=0)
            MoveDirectionNode (selectedDirection=ZPlus toolParams=0.02, 0.02)
              Until DISTANCE (allowActions=false deceleration=3 distanceNodeType=STOP) Distance=0.075; motionParameters(blendRadius=0)
        Folder Buje3
          Xfin := ((0.14605*Xp)-(Xd)-(0.3937*(1/m2)))*(-1)
          Yfin := ((0.3937*Yp)-(Yd)+(0.14605*m1))*(-1)
          rotaciones := get_actual_tcp_pose()
          var_3 := rotaciones[3]
          var_4 := rotaciones[4]
          var_5 := rotaciones[5]
          PosFinal := p[Xfin+0.00208915,Yfin+0.00208915,-0.440,var_3,var_4,var_5]
          MoveL speed 250 mm/s, acceleration 1200 mm/s^2 (useActiveTCP=true) feature=Base
            MoveJ speed 60 deg/s, acceleration 80 deg/s^2 (useActiveTCP=true) feature=Base
              Waypoint Waypoint (Variable): motionParameters(jointSpeed=1.047198 jointAcceleration=1.396263 cartesianSpeed=0.15 cartesianAcceleration=0.2); variable=PosFinal
            MoveDirectionNode (selectedDirection=ZMinus toolParams=0.02, 0.02)
              Until DISTANCE (allowActions=false deceleration=3 distanceNodeType=STOP) Distance=0.075; motionParameters(blendRadius=0)
            MoveDirectionNode (selectedDirection=ZPlus toolParams=0.02, 0.02)
              Until DISTANCE (allowActions=false deceleration=3 distanceNodeType=STOP) Distance=0.075; motionParameters(blendRadius=0)
        Folder Buje4
          Xfin := ((0.17145*Xp)-(Xd)-(0.3937*(1/m2)))*(-1)
          Yfin := ((0.3937*Yp)-(Yd)+(0.17145*m1))*(-1)
          rotaciones := get_actual_tcp_pose()
          var_3 := rotaciones[3]
          var_4 := rotaciones[4]
          var_5 := rotaciones[5]
          PosFinal := p[Xfin+0.00208915,Yfin+0.00208915,-0.44,var_3,var_4,var_5]
          MoveL speed 250 mm/s, acceleration 1200 mm/s^2 (useActiveTCP=true) feature=Base
            MoveJ speed 60 deg/s, acceleration 80 deg/s^2 (useActiveTCP=true) feature=Base
              Waypoint Waypoint (Variable): motionParameters(jointSpeed=1.047198 jointAcceleration=1.396263 cartesianSpeed=0.15 cartesianAcceleration=0.2); variable=PosFinal
            MoveDirectionNode (selectedDirection=ZMinus toolParams=0.02, 0.02)
              Until DISTANCE (allowActions=false deceleration=3 distanceNodeType=STOP) Distance=0.075; motionParameters(blendRadius=0)
            MoveDirectionNode (selectedDirection=ZPlus toolParams=0.02, 0.02)
              Until DISTANCE (allowActions=false deceleration=3 distanceNodeType=STOP) Distance=0.075; motionParameters(blendRadius=0)
        Folder Buje5
          Xfin := ((0.19685*Xp)-(Xd)-(0.3937*(1/m2)))*(-1)
          Yfin := ((0.3937*Yp)-(Yd)+(0.19685*m1))*(-1)
          rotaciones := get_actual_tcp_pose()
          var_3 := rotaciones[3]
          var_4 := rotaciones[4]
          var_5 := rotaciones[5]
          PosFinal := p[Xfin+0.00208915,Yfin+0.00208915,-0.44,var_3,var_4,var_5]
          MoveL speed 250 mm/s, acceleration 1200 mm/s^2 (useActiveTCP=true) feature=Base
            MoveJ speed 60 deg/s, acceleration 80 deg/s^2 (useActiveTCP=true) feature=Base
              Waypoint Waypoint (Variable): motionParameters(jointSpeed=1.047198 jointAcceleration=1.396263 cartesianSpeed=0.15 cartesianAcceleration=0.2); variable=PosFinal
            MoveDirectionNode (selectedDirection=ZMinus toolParams=0.02, 0.02)
              Until DISTANCE (allowActions=false deceleration=3 distanceNodeType=STOP) Distance=0.075; motionParameters(blendRadius=0)
            MoveDirectionNode (selectedDirection=ZPlus toolParams=0.02, 0.02)
              Until DISTANCE (allowActions=false deceleration=3 distanceNodeType=STOP) Distance=0.075; motionParameters(blendRadius=0)
        Folder Buje6
          Xfin := ((0.22225*Xp)-(Xd)-(0.3937*(1/m2)))*(-1)
          Yfin := ((0.3937*Yp)-(Yd)+(0.22225*m1))*(-1)
          rotaciones := get_actual_tcp_pose()
          var_3 := rotaciones[3]
          var_4 := rotaciones[4]
          var_5 := rotaciones[5]
          PosFinal := p[Xfin+0.00208915,Yfin+0.00208915,-0.44,var_3,var_4,var_5]
          MoveL speed 250 mm/s, acceleration 1200 mm/s^2 (useActiveTCP=true) feature=Base
            MoveJ speed 60 deg/s, acceleration 80 deg/s^2 (useActiveTCP=true) feature=Base
              Waypoint Waypoint (Variable): motionParameters(jointSpeed=1.047198 jointAcceleration=1.396263 cartesianSpeed=0.15 cartesianAcceleration=0.2); variable=PosFinal
            MoveDirectionNode (selectedDirection=ZMinus toolParams=0.02, 0.02)
              Until DISTANCE (allowActions=false deceleration=3 distanceNodeType=STOP) Distance=0.075; motionParameters(blendRadius=0)
            MoveDirectionNode (selectedDirection=ZPlus toolParams=0.02, 0.02)
              Until DISTANCE (allowActions=false deceleration=3 distanceNodeType=STOP) Distance=0.075; motionParameters(blendRadius=0)
        Folder Buje7
          Xfin := ((0.24765*Xp)-(Xd)-(0.3937*(1/m2)))*(-1)
          Yfin := ((0.3937*Yp)-(Yd)+(0.24765*m1))*(-1)
          rotaciones := get_actual_tcp_pose()
          var_3 := rotaciones[3]
          var_4 := rotaciones[4]
          var_5 := rotaciones[5]
          PosFinal := p[Xfin+0.00208915,Yfin+0.00208915,-0.44,var_3,var_4,var_5]
          MoveL speed 250 mm/s, acceleration 1200 mm/s^2 (useActiveTCP=true) feature=Base
            MoveJ speed 60 deg/s, acceleration 80 deg/s^2 (useActiveTCP=true) feature=Base
              Waypoint Waypoint (Variable): motionParameters(jointSpeed=1.047198 jointAcceleration=1.396263 cartesianSpeed=0.15 cartesianAcceleration=0.2); variable=PosFinal
            MoveDirectionNode (selectedDirection=ZMinus toolParams=0.02, 0.02)
              Until DISTANCE (allowActions=false deceleration=3 distanceNodeType=STOP) Distance=0.075; motionParameters(blendRadius=0)
            MoveDirectionNode (selectedDirection=ZPlus toolParams=0.02, 0.02)
              Until DISTANCE (allowActions=false deceleration=3 distanceNodeType=STOP) Distance=0.075; motionParameters(blendRadius=0)
        Folder Buje8
          Xfin := ((0.27305*Xp)-(Xd)-(0.3937*(1/m2)))*(-1)
          Yfin := ((0.3937*Yp)-(Yd)+(0.27305*m1))*(-1)
          rotaciones := get_actual_tcp_pose()
          var_3 := rotaciones[3]
          var_4 := rotaciones[4]
          var_5 := rotaciones[5]
          PosFinal := p[Xfin+0.00208915,Yfin+0.00208915,-0.44,var_3,var_4,var_5]
          MoveL speed 250 mm/s, acceleration 1200 mm/s^2 (useActiveTCP=true) feature=Base
            MoveJ speed 60 deg/s, acceleration 80 deg/s^2 (useActiveTCP=true) feature=Base
              Waypoint Waypoint (Variable): motionParameters(jointSpeed=1.047198 jointAcceleration=1.396263 cartesianSpeed=0.15 cartesianAcceleration=0.2); variable=PosFinal
            MoveDirectionNode (selectedDirection=ZMinus toolParams=0.02, 0.02)
              Until DISTANCE (allowActions=false deceleration=3 distanceNodeType=STOP) Distance=0.075; motionParameters(blendRadius=0)
            MoveDirectionNode (selectedDirection=ZPlus toolParams=0.02, 0.02)
              Until DISTANCE (allowActions=false deceleration=3 distanceNodeType=STOP) Distance=0.075; motionParameters(blendRadius=0)
        Folder Buje9
          Xfin := ((0.29845*Xp)-(Xd)-(0.3937*(1/m2)))*(-1)
          Yfin := ((0.3937*Yp)-(Yd)+(0.29845*m1))*(-1)
          rotaciones := get_actual_tcp_pose()
          var_3 := rotaciones[3]
          var_4 := rotaciones[4]
          var_5 := rotaciones[5]
          PosFinal := p[Xfin+0.00208915,Yfin+0.00208915,-0.44,var_3,var_4,var_5]
          MoveL speed 250 mm/s, acceleration 1200 mm/s^2 (useActiveTCP=true) feature=Base
            MoveJ speed 60 deg/s, acceleration 80 deg/s^2 (useActiveTCP=true) feature=Base
              Waypoint Waypoint (Variable): motionParameters(jointSpeed=1.047198 jointAcceleration=1.396263 cartesianSpeed=0.15 cartesianAcceleration=0.2); variable=PosFinal
            MoveDirectionNode (selectedDirection=ZMinus toolParams=0.02, 0.02)
              Until DISTANCE (allowActions=false deceleration=3 distanceNodeType=STOP) Distance=0.075; motionParameters(blendRadius=0)
            MoveDirectionNode (selectedDirection=ZPlus toolParams=0.02, 0.02)
              Until DISTANCE (allowActions=false deceleration=3 distanceNodeType=STOP) Distance=0.075; motionParameters(blendRadius=0)
        Folder Buje10
          Xfin := ((0.32385*Xp)-(Xd)-(0.3937*(1/m2)))*(-1)
          Yfin := ((0.3937*Yp)-(Yd)+(0.32385*m1))*(-1)
          rotaciones := get_actual_tcp_pose()
          var_3 := rotaciones[3]
          var_4 := rotaciones[4]
          var_5 := rotaciones[5]
          PosFinal := p[Xfin+0.00208915,Yfin+0.00208915,-0.44,var_3,var_4,var_5]
          MoveL speed 250 mm/s, acceleration 1200 mm/s^2 (useActiveTCP=true) feature=Base
            MoveJ speed 60 deg/s, acceleration 80 deg/s^2 (useActiveTCP=true) feature=Base
              Waypoint Waypoint (Variable): motionParameters(jointSpeed=1.047198 jointAcceleration=1.396263 cartesianSpeed=0.15 cartesianAcceleration=0.2); variable=PosFinal
            MoveDirectionNode (selectedDirection=ZMinus toolParams=0.02, 0.02)
              Until DISTANCE (allowActions=false deceleration=3 distanceNodeType=STOP) Distance=0.075; motionParameters(blendRadius=0)
            MoveDirectionNode (selectedDirection=ZPlus toolParams=0.02, 0.02)
              Until DISTANCE (allowActions=false deceleration=3 distanceNodeType=STOP) Distance=0.075; motionParameters(blendRadius=0)
        Folder Buje11
          Xfin := ((0.34925*Xp)-(Xd)-(0.3937*(1/m2)))*(-1)
          Yfin := ((0.3937*Yp)-(Yd)+(0.34925*m1))*(-1)
          rotaciones := get_actual_tcp_pose()
          var_3 := rotaciones[3]
          var_4 := rotaciones[4]
          var_5 := rotaciones[5]
          PosFinal := p[Xfin+0.00208915,Yfin+0.00208915,-0.44,var_3,var_4,var_5]
          MoveL speed 250 mm/s, acceleration 1200 mm/s^2 (useActiveTCP=true) feature=Base
            MoveJ speed 60 deg/s, acceleration 80 deg/s^2 (useActiveTCP=true) feature=Base
              Waypoint Waypoint (Variable): motionParameters(jointSpeed=1.047198 jointAcceleration=1.396263 cartesianSpeed=0.15 cartesianAcceleration=0.2); variable=PosFinal
            MoveDirectionNode (selectedDirection=ZMinus toolParams=0.02, 0.02)
              Until DISTANCE (allowActions=false deceleration=3 distanceNodeType=STOP) Distance=0.075; motionParameters(blendRadius=0)
            MoveDirectionNode (selectedDirection=ZPlus toolParams=0.02, 0.02)
              Until DISTANCE (allowActions=false deceleration=3 distanceNodeType=STOP) Distance=0.075; motionParameters(blendRadius=0)
        Folder Buje12
          Xfin := ((0.37465*Xp)-(Xd)-(0.3937*(1/m2)))*(-1)
          Yfin := ((0.3937*Yp)-(Yd)+(0.37465*m1))*(-1)
          rotaciones := get_actual_tcp_pose()
          var_3 := rotaciones[3]
          var_4 := rotaciones[4]
          var_5 := rotaciones[5]
          PosFinal := p[Xfin+0.00208915,Yfin+0.00208915,-0.44,var_3,var_4,var_5]
          MoveL speed 250 mm/s, acceleration 1200 mm/s^2 (useActiveTCP=true) feature=Base
            MoveJ speed 60 deg/s, acceleration 80 deg/s^2 (useActiveTCP=true) feature=Base
              Waypoint Waypoint (Variable): motionParameters(jointSpeed=1.047198 jointAcceleration=1.396263 cartesianSpeed=0.15 cartesianAcceleration=0.2); variable=PosFinal
            MoveDirectionNode (selectedDirection=ZMinus toolParams=0.02, 0.02)
              Until DISTANCE (allowActions=false deceleration=3 distanceNodeType=STOP) Distance=0.075; motionParameters(blendRadius=0)
            MoveDirectionNode (selectedDirection=ZPlus toolParams=0.02, 0.02)
              Until DISTANCE (allowActions=false deceleration=3 distanceNodeType=STOP) Distance=0.075; motionParameters(blendRadius=0)
        Folder Buje13
          Xfin := ((0.40005*Xp)-(Xd)-(0.3937*(1/m2)))*(-1)
          Yfin := ((0.3937*Yp)-(Yd)+(0.40005*m1))*(-1)
          rotaciones := get_actual_tcp_pose()
          var_3 := rotaciones[3]
          var_4 := rotaciones[4]
          var_5 := rotaciones[5]
          PosFinal := p[Xfin+0.00208915,Yfin+0.00208915,-0.44,var_3,var_4,var_5]
          MoveL speed 250 mm/s, acceleration 1200 mm/s^2 (useActiveTCP=true) feature=Base
            MoveJ speed 60 deg/s, acceleration 80 deg/s^2 (useActiveTCP=true) feature=Base
              Waypoint Waypoint (Variable): motionParameters(jointSpeed=1.047198 jointAcceleration=1.396263 cartesianSpeed=0.15 cartesianAcceleration=0.2); variable=PosFinal
            MoveDirectionNode (selectedDirection=ZMinus toolParams=0.02, 0.02)
              Until DISTANCE (allowActions=false deceleration=3 distanceNodeType=STOP) Distance=0.075; motionParameters(blendRadius=0)
            MoveDirectionNode (selectedDirection=ZPlus toolParams=0.02, 0.02)
              Until DISTANCE (allowActions=false deceleration=3 distanceNodeType=STOP) Distance=0.075; motionParameters(blendRadius=0)
        Folder Buje14
          Xfin := ((0.42545*Xp)-(Xd)-(0.3937*(1/m2)))*(-1)
          Yfin := ((0.3937*Yp)-(Yd)+(0.42545*m1))*(-1)
          rotaciones := get_actual_tcp_pose()
          var_3 := rotaciones[3]
          var_4 := rotaciones[4]
          var_5 := rotaciones[5]
          PosFinal := p[Xfin+0.00208915,Yfin+0.00208915,-0.44,var_3,var_4,var_5]
          MoveL speed 250 mm/s, acceleration 1200 mm/s^2 (useActiveTCP=true) feature=Base
            MoveJ speed 60 deg/s, acceleration 80 deg/s^2 (useActiveTCP=true) feature=Base
              Waypoint Waypoint (Variable): motionParameters(jointSpeed=1.047198 jointAcceleration=1.396263 cartesianSpeed=0.15 cartesianAcceleration=0.2); variable=PosFinal
            MoveDirectionNode (selectedDirection=ZMinus toolParams=0.02, 0.02)
              Until DISTANCE (allowActions=false deceleration=3 distanceNodeType=STOP) Distance=0.075; motionParameters(blendRadius=0)
            MoveDirectionNode (selectedDirection=ZPlus toolParams=0.02, 0.02)
              Until DISTANCE (allowActions=false deceleration=3 distanceNodeType=STOP) Distance=0.075; motionParameters(blendRadius=0)
        Folder Buje15
          Xfin := ((0.45085*Xp)-(Xd)-(0.3937*(1/m2)))*(-1)
          Yfin := ((0.3937*Yp)-(Yd)+(0.45085*m1))*(-1)
          rotaciones := get_actual_tcp_pose()
          var_3 := rotaciones[3]
          var_4 := rotaciones[4]
          var_5 := rotaciones[5]
          PosFinal := p[Xfin+0.00208915,Yfin+0.00208915,-0.44,var_3,var_4,var_5]
          MoveL speed 250 mm/s, acceleration 1200 mm/s^2 (useActiveTCP=true) feature=Base
            MoveJ speed 60 deg/s, acceleration 80 deg/s^2 (useActiveTCP=true) feature=Base
              Waypoint Waypoint (Variable): motionParameters(jointSpeed=1.047198 jointAcceleration=1.396263 cartesianSpeed=0.15 cartesianAcceleration=0.2); variable=PosFinal
            MoveDirectionNode (selectedDirection=ZMinus toolParams=0.02, 0.02)
              Until DISTANCE (allowActions=false deceleration=3 distanceNodeType=STOP) Distance=0.075; motionParameters(blendRadius=0)
            MoveDirectionNode (selectedDirection=ZPlus toolParams=0.02, 0.02)
              Until DISTANCE (allowActions=false deceleration=3 distanceNodeType=STOP) Distance=0.075; motionParameters(blendRadius=0)
        Folder Buje16
          Xfin := ((0.47625*Xp)-(Xd)-(0.3937*(1/m2)))*(-1)
          Yfin := ((0.3937*Yp)-(Yd)+(0.47625*m1))*(-1)
          rotaciones := get_actual_tcp_pose()
          var_3 := rotaciones[3]
          var_4 := rotaciones[4]
          var_5 := rotaciones[5]
          PosFinal := p[Xfin+0.00208915,Yfin+0.00208915,-0.44,var_3,var_4,var_5]
          MoveL speed 250 mm/s, acceleration 1200 mm/s^2 (useActiveTCP=true) feature=Base
            MoveJ speed 60 deg/s, acceleration 80 deg/s^2 (useActiveTCP=true) feature=Base
              Waypoint Waypoint (Variable): motionParameters(jointSpeed=1.047198 jointAcceleration=1.396263 cartesianSpeed=0.15 cartesianAcceleration=0.2); variable=PosFinal
            MoveDirectionNode (selectedDirection=ZMinus toolParams=0.02, 0.02)
              Until DISTANCE (allowActions=false deceleration=3 distanceNodeType=STOP) Distance=0.075; motionParameters(blendRadius=0)
            MoveDirectionNode (selectedDirection=ZPlus toolParams=0.02, 0.02)
              Until DISTANCE (allowActions=false deceleration=3 distanceNodeType=STOP) Distance=0.075; motionParameters(blendRadius=0)
        Folder Buje17
          Xfin := ((0.50165*Xp)-(Xd)-(0.3937*(1/m2)))*(-1)
          Yfin := ((0.3937*Yp)-(Yd)+(0.50165*m1))*(-1)
          rotaciones := get_actual_tcp_pose()
          var_3 := rotaciones[3]
          var_4 := rotaciones[4]
          var_5 := rotaciones[5]
          PosFinal := p[Xfin+0.00208915,Yfin+0.00208915,-0.44,var_3,var_4,var_5]
          MoveL speed 250 mm/s, acceleration 1200 mm/s^2 (useActiveTCP=true) feature=Base
            MoveJ speed 60 deg/s, acceleration 80 deg/s^2 (useActiveTCP=true) feature=Base
              Waypoint Waypoint (Variable): motionParameters(jointSpeed=1.047198 jointAcceleration=1.396263 cartesianSpeed=0.15 cartesianAcceleration=0.2); variable=PosFinal
            MoveDirectionNode (selectedDirection=ZMinus toolParams=0.02, 0.02)
              Until DISTANCE (allowActions=false deceleration=3 distanceNodeType=STOP) Distance=0.075; motionParameters(blendRadius=0)
            MoveDirectionNode (selectedDirection=ZPlus toolParams=0.02, 0.02)
              Until DISTANCE (allowActions=false deceleration=3 distanceNodeType=STOP) Distance=0.075; motionParameters(blendRadius=0)
        Folder Buje18
          Xfin := ((0.52705*Xp)-(Xd)-(0.3937*(1/m2)))*(-1)
          Yfin := ((0.3937*Yp)-(Yd)+(0.52705*m1))*(-1)
          rotaciones := get_actual_tcp_pose()
          var_3 := rotaciones[3]
          var_4 := rotaciones[4]
          var_5 := rotaciones[5]
          PosFinal := p[Xfin+0.00208915,Yfin+0.00208915,-0.44,var_3,var_4,var_5]
          MoveL speed 250 mm/s, acceleration 1200 mm/s^2 (useActiveTCP=true) feature=Base
            MoveJ speed 60 deg/s, acceleration 80 deg/s^2 (useActiveTCP=true) feature=Base
              Waypoint Waypoint (Variable): motionParameters(jointSpeed=1.047198 jointAcceleration=1.396263 cartesianSpeed=0.15 cartesianAcceleration=0.2); variable=PosFinal
            MoveDirectionNode (selectedDirection=ZMinus toolParams=0.02, 0.02)
              Until DISTANCE (allowActions=false deceleration=3 distanceNodeType=STOP) Distance=0.075; motionParameters(blendRadius=0)
            MoveDirectionNode (selectedDirection=ZPlus toolParams=0.02, 0.02)
              Until DISTANCE (allowActions=false deceleration=3 distanceNodeType=STOP) Distance=0.075; motionParameters(blendRadius=0)
        Folder Buje19
          Xfin := ((0.55245*Xp)-(Xd)-(0.3937*(1/m2)))*(-1)
          Yfin := ((0.3937*Yp)-(Yd)+(0.55245*m1))*(-1)
          rotaciones := get_actual_tcp_pose()
          var_3 := rotaciones[3]
          var_4 := rotaciones[4]
          var_5 := rotaciones[5]
          PosFinal := p[Xfin+0.00208915,Yfin+0.00208915,-0.44,var_3,var_4,var_5]
          MoveL speed 250 mm/s, acceleration 1200 mm/s^2 (useActiveTCP=true) feature=Base
            MoveJ speed 60 deg/s, acceleration 80 deg/s^2 (useActiveTCP=true) feature=Base
              Waypoint Waypoint (Variable): motionParameters(jointSpeed=1.047198 jointAcceleration=1.396263 cartesianSpeed=0.15 cartesianAcceleration=0.2); variable=PosFinal
            MoveDirectionNode (selectedDirection=ZMinus toolParams=0.02, 0.02)
              Until DISTANCE (allowActions=false deceleration=3 distanceNodeType=STOP) Distance=0.075; motionParameters(blendRadius=0)
            MoveDirectionNode (selectedDirection=ZPlus toolParams=0.02, 0.02)
              Until DISTANCE (allowActions=false deceleration=3 distanceNodeType=STOP) Distance=0.075; motionParameters(blendRadius=0)
        Folder Buje20
          Xfin := ((0.57785*Xp)-(Xd)-(0.3937*(1/m2)))*(-1)
          Yfin := ((0.3937*Yp)-(Yd)+(0.57785*m1))*(-1)
          rotaciones := get_actual_tcp_pose()
          var_3 := rotaciones[3]
          var_4 := rotaciones[4]
          var_5 := rotaciones[5]
          PosFinal := p[Xfin+0.00208915,Yfin+0.00208915,-0.44,var_3,var_4,var_5]
          MoveL speed 250 mm/s, acceleration 1200 mm/s^2 (useActiveTCP=true) feature=Base
            MoveJ speed 60 deg/s, acceleration 80 deg/s^2 (useActiveTCP=true) feature=Base
              Waypoint Waypoint (Variable): motionParameters(jointSpeed=1.047198 jointAcceleration=1.396263 cartesianSpeed=0.15 cartesianAcceleration=0.2); variable=PosFinal
            MoveDirectionNode (selectedDirection=ZMinus toolParams=0.02, 0.02)
              Until DISTANCE (allowActions=false deceleration=3 distanceNodeType=STOP) Distance=0.075; motionParameters(blendRadius=0)
            MoveDirectionNode (selectedDirection=ZPlus toolParams=0.02, 0.02)
              Until DISTANCE (allowActions=false deceleration=3 distanceNodeType=STOP) Distance=0.075; motionParameters(blendRadius=0)
        Folder Buje21
          Xfin := ((0.60325*Xp)-(Xd)-(0.3937*(1/m2)))*(-1)
          Yfin := ((0.3937*Yp)-(Yd)+(0.60325*m1))*(-1)
          rotaciones := get_actual_tcp_pose()
          var_3 := rotaciones[3]
          var_4 := rotaciones[4]
          var_5 := rotaciones[5]
          PosFinal := p[Xfin+0.00208915,Yfin+0.00208915,-0.44,var_3,var_4,var_5]
          MoveL speed 250 mm/s, acceleration 1200 mm/s^2 (useActiveTCP=true) feature=Base
            MoveJ speed 60 deg/s, acceleration 80 deg/s^2 (useActiveTCP=true) feature=Base
              Waypoint Waypoint (Variable): motionParameters(jointSpeed=1.047198 jointAcceleration=1.396263 cartesianSpeed=0.15 cartesianAcceleration=0.2); variable=PosFinal
            MoveDirectionNode (selectedDirection=ZMinus toolParams=0.02, 0.02)
              Until DISTANCE (allowActions=false deceleration=3 distanceNodeType=STOP) Distance=0.075; motionParameters(blendRadius=0)
            MoveDirectionNode (selectedDirection=ZPlus toolParams=0.02, 0.02)
              Until DISTANCE (allowActions=false deceleration=3 distanceNodeType=STOP) Distance=0.075; motionParameters(blendRadius=0)
        Folder Buje22
          Xfin := ((0.62865*Xp)-(Xd)-(0.3937*(1/m2)))*(-1)
          Yfin := ((0.3937*Yp)-(Yd)+(0.62865*m1))*(-1)
          rotaciones := get_actual_tcp_pose()
          var_3 := rotaciones[3]
          var_4 := rotaciones[4]
          var_5 := rotaciones[5]
          PosFinal := p[Xfin+0.00208915,Yfin+0.00208915,-0.44,var_3,var_4,var_5]
          MoveL speed 250 mm/s, acceleration 1200 mm/s^2 (useActiveTCP=true) feature=Base
            MoveJ speed 60 deg/s, acceleration 80 deg/s^2 (useActiveTCP=true) feature=Base
              Waypoint Waypoint (Variable): motionParameters(jointSpeed=1.047198 jointAcceleration=1.396263 cartesianSpeed=0.15 cartesianAcceleration=0.2); variable=PosFinal
            MoveDirectionNode (selectedDirection=ZMinus toolParams=0.02, 0.02)
              Until DISTANCE (allowActions=false deceleration=3 distanceNodeType=STOP) Distance=0.075; motionParameters(blendRadius=0)
            MoveDirectionNode (selectedDirection=ZPlus toolParams=0.02, 0.02)
              Until DISTANCE (allowActions=false deceleration=3 distanceNodeType=STOP) Distance=0.075; motionParameters(blendRadius=0)
        Folder Buje23
          Xfin := ((0.65405*Xp)-(Xd)-(0.3937*(1/m2)))*(-1)
          Yfin := ((0.3937*Yp)-(Yd)+(0.65405*m1))*(-1)
          rotaciones := get_actual_tcp_pose()
          var_3 := rotaciones[3]
          var_4 := rotaciones[4]
          var_5 := rotaciones[5]
          PosFinal := p[Xfin+0.00208915,Yfin+0.00208915,-0.44,var_3,var_4,var_5]
          MoveL speed 250 mm/s, acceleration 1200 mm/s^2 (useActiveTCP=true) feature=Base
            MoveJ speed 60 deg/s, acceleration 80 deg/s^2 (useActiveTCP=true) feature=Base
              Waypoint Waypoint (Variable): motionParameters(jointSpeed=1.047198 jointAcceleration=1.396263 cartesianSpeed=0.15 cartesianAcceleration=0.2); variable=PosFinal
            MoveDirectionNode (selectedDirection=ZMinus toolParams=0.02, 0.02)
              Until DISTANCE (allowActions=false deceleration=3 distanceNodeType=STOP) Distance=0.075; motionParameters(blendRadius=0)
            MoveDirectionNode (selectedDirection=ZPlus toolParams=0.02, 0.02)
              Until DISTANCE (allowActions=false deceleration=3 distanceNodeType=STOP) Distance=0.075; motionParameters(blendRadius=0)
        Folder Buje24
          Xfin := ((0.67945*Xp)-(Xd)-(0.3937*(1/m2)))*(-1)
          Yfin := ((0.3937*Yp)-(Yd)+(0.67945*m1))*(-1)
          rotaciones := get_actual_tcp_pose()
          var_3 := rotaciones[3]
          var_4 := rotaciones[4]
          var_5 := rotaciones[5]
          PosFinal := p[Xfin+0.00208915,Yfin+0.00208915,-0.44,var_3,var_4,var_5]
          MoveL speed 250 mm/s, acceleration 1200 mm/s^2 (useActiveTCP=true) feature=Base
            MoveJ speed 60 deg/s, acceleration 80 deg/s^2 (useActiveTCP=true) feature=Base
              Waypoint Waypoint (Variable): motionParameters(jointSpeed=1.047198 jointAcceleration=1.396263 cartesianSpeed=0.15 cartesianAcceleration=0.2); variable=PosFinal
            MoveDirectionNode (selectedDirection=ZMinus toolParams=0.02, 0.02)
              Until DISTANCE (allowActions=false deceleration=3 distanceNodeType=STOP) Distance=0.075; motionParameters(blendRadius=0)
            MoveDirectionNode (selectedDirection=ZPlus toolParams=0.02, 0.02)
              Until DISTANCE (allowActions=false deceleration=3 distanceNodeType=STOP) Distance=0.075; motionParameters(blendRadius=0)
        Folder Buje25
          Xfin := ((0.70485*Xp)-(Xd)-(0.3937*(1/m2)))*(-1)
          Yfin := ((0.3937*Yp)-(Yd)+(0.70485*m1))*(-1)
          rotaciones := get_actual_tcp_pose()
          var_3 := rotaciones[3]
          var_4 := rotaciones[4]
          var_5 := rotaciones[5]
          PosFinal := p[Xfin+0.00208915,Yfin+0.00208915,-0.44,var_3,var_4,var_5]
          MoveL speed 250 mm/s, acceleration 1200 mm/s^2 (useActiveTCP=true) feature=Base
            MoveJ speed 60 deg/s, acceleration 80 deg/s^2 (useActiveTCP=true) feature=Base
              Waypoint Waypoint (Variable): motionParameters(jointSpeed=1.047198 jointAcceleration=1.396263 cartesianSpeed=0.15 cartesianAcceleration=0.2); variable=PosFinal
            MoveDirectionNode (selectedDirection=ZMinus toolParams=0.02, 0.02)
              Until DISTANCE (allowActions=false deceleration=3 distanceNodeType=STOP) Distance=0.075; motionParameters(blendRadius=0)
            MoveDirectionNode (selectedDirection=ZPlus toolParams=0.02, 0.02)
              Until DISTANCE (allowActions=false deceleration=3 distanceNodeType=STOP) Distance=0.075; motionParameters(blendRadius=0)
        Folder Buje26
          Xfin := ((0.73025*Xp)-(Xd)-(0.3937*(1/m2)))*(-1)
          Yfin := ((0.3937*Yp)-(Yd)+(0.73025*m1))*(-1)
          rotaciones := get_actual_tcp_pose()
          var_3 := rotaciones[3]
          var_4 := rotaciones[4]
          var_5 := rotaciones[5]
          PosFinal := p[Xfin+0.00208915,Yfin+0.00208915,-0.44,var_3,var_4,var_5]
          MoveL speed 250 mm/s, acceleration 1200 mm/s^2 (useActiveTCP=true) feature=Base
            MoveJ speed 60 deg/s, acceleration 80 deg/s^2 (useActiveTCP=true) feature=Base
              Waypoint Waypoint (Variable): motionParameters(jointSpeed=1.047198 jointAcceleration=1.396263 cartesianSpeed=0.15 cartesianAcceleration=0.2); variable=PosFinal
            MoveDirectionNode (selectedDirection=ZMinus toolParams=0.02, 0.02)
              Until DISTANCE (allowActions=false deceleration=3 distanceNodeType=STOP) Distance=0.075; motionParameters(blendRadius=0)
            MoveDirectionNode (selectedDirection=ZPlus toolParams=0.02, 0.02)
              Until DISTANCE (allowActions=false deceleration=3 distanceNodeType=STOP) Distance=0.075; motionParameters(blendRadius=0)
        Folder Buje27
          Xfin := ((0.75565*Xp)-(Xd)-(0.3937*(1/m2)))*(-1)
          Yfin := ((0.3937*Yp)-(Yd)+(0.75565*m1))*(-1)
          rotaciones := get_actual_tcp_pose()
          var_3 := rotaciones[3]
          var_4 := rotaciones[4]
          var_5 := rotaciones[5]
          PosFinal := p[Xfin+0.00208915,Yfin+0.00208915,-0.44,var_3,var_4,var_5]
          MoveL speed 250 mm/s, acceleration 1200 mm/s^2 (useActiveTCP=true) feature=Base
            MoveJ speed 60 deg/s, acceleration 80 deg/s^2 (useActiveTCP=true) feature=Base
              Waypoint Waypoint (Variable): motionParameters(jointSpeed=1.047198 jointAcceleration=1.396263 cartesianSpeed=0.15 cartesianAcceleration=0.2); variable=PosFinal
            MoveDirectionNode (selectedDirection=ZMinus toolParams=0.02, 0.02)
              Until DISTANCE (allowActions=false deceleration=3 distanceNodeType=STOP) Distance=0.075; motionParameters(blendRadius=0)
            MoveDirectionNode (selectedDirection=ZPlus toolParams=0.02, 0.02)
              Until DISTANCE (allowActions=false deceleration=3 distanceNodeType=STOP) Distance=0.075; motionParameters(blendRadius=0)
SubProgram GoNoGo (keepSynchronizedWithDisk=false)
  Folder GoNoGo
    Folder Buje1
      Xfin := ((0.09525*Xp)-(Xd)-(-0.0127*(1/m2)))*(-1)
      Yfin := ((-0.0127*Yp)-(Yd)+(0.09525*m1))*(-1)
      rotaciones := get_actual_tcp_pose()
      var_3 := rotaciones[3]
      var_4 := rotaciones[4]
      var_5 := rotaciones[5]
      PosFinal := p[Xfin+0.00208915,Yfin+0.00208915,0.11,var_3,var_4,var_5]
      MoveL speed 250 mm/s, acceleration 1200 mm/s^2 (useActiveTCP=true) feature=Base
        MoveJ speed 60 deg/s, acceleration 80 deg/s^2 (useActiveTCP=true) feature=Base
          Waypoint Waypoint (Variable): motionParameters(jointSpeed=1.047198 jointAcceleration=1.396263 cartesianSpeed=0.15 cartesianAcceleration=0.2); variable=PosFinal
        MoveDirectionNode (selectedDirection=ZMinus toolParams=0.02, 0.02)
          Until DISTANCE (allowActions=false deceleration=3 distanceNodeType=STOP) Distance=0.075; motionParameters(blendRadius=0)
        MoveDirectionNode (selectedDirection=ZPlus toolParams=0.02, 0.02)
          Until DISTANCE (allowActions=false deceleration=3 distanceNodeType=STOP) Distance=0.075; motionParameters(blendRadius=0)
    Folder Buje2
      Xfin := ((0.12065*Xp)-(Xd)-(-0.0127*(1/m2)))*(-1)
      Yfin := ((-0.0127*Yp)-(Yd)+(0.12065*m1))*(-1)
      rotaciones := get_actual_tcp_pose()
      var_3 := rotaciones[3]
      var_4 := rotaciones[4]
      var_5 := rotaciones[5]
      PosFinal := p[Xfin+0.00208915,Yfin+0.00208915,0.11,var_3,var_4,var_5]
      MoveL speed 250 mm/s, acceleration 1200 mm/s^2 (useActiveTCP=true) feature=Base
        MoveJ speed 60 deg/s, acceleration 80 deg/s^2 (useActiveTCP=true) feature=Base
          Waypoint Waypoint (Variable): motionParameters(jointSpeed=1.047198 jointAcceleration=1.396263 cartesianSpeed=0.15 cartesianAcceleration=0.2); variable=PosFinal
        MoveDirectionNode (selectedDirection=ZMinus toolParams=0.02, 0.02)
          Until DISTANCE (allowActions=false deceleration=3 distanceNodeType=STOP) Distance=0.075; motionParameters(blendRadius=0)
        MoveDirectionNode (selectedDirection=ZPlus toolParams=0.02, 0.02)
          Until DISTANCE (allowActions=false deceleration=3 distanceNodeType=STOP) Distance=0.075; motionParameters(blendRadius=0)
    Folder Buje3
      Xfin := ((0.14605*Xp)-(Xd)-(-0.0127*(1/m2)))*(-1)
      Yfin := ((-0.0127*Yp)-(Yd)+(0.14605*m1))*(-1)
      rotaciones := get_actual_tcp_pose()
      var_3 := rotaciones[3]
      var_4 := rotaciones[4]
      var_5 := rotaciones[5]
      PosFinal := p[Xfin+0.00208915,Yfin+0.00208915,0.11,var_3,var_4,var_5]
      MoveL speed 250 mm/s, acceleration 1200 mm/s^2 (useActiveTCP=true) feature=Base
        MoveJ speed 60 deg/s, acceleration 80 deg/s^2 (useActiveTCP=true) feature=Base
          Waypoint Waypoint (Variable): motionParameters(jointSpeed=1.047198 jointAcceleration=1.396263 cartesianSpeed=0.15 cartesianAcceleration=0.2); variable=PosFinal
        MoveDirectionNode (selectedDirection=ZMinus toolParams=0.02, 0.02)
          Until DISTANCE (allowActions=false deceleration=3 distanceNodeType=STOP) Distance=0.075; motionParameters(blendRadius=0)
        MoveDirectionNode (selectedDirection=ZPlus toolParams=0.02, 0.02)
          Until DISTANCE (allowActions=false deceleration=3 distanceNodeType=STOP) Distance=0.075; motionParameters(blendRadius=0)
